FUNCTION_BLOCK TestSuite
VAR_GENERIC CONSTANT
	_MaxTestCount : DINT := 10;
END_VAR IMPLEMENTS I_TestSuite
VAR
	_TestSuiteName	  : STRING;
	TestCollection	  : ARRAY[0.._MaxTestCount] OF Test;
	NoAction		  : Test := (TestId := 'No Action', State := E_TestStatus.DoneOk);
	ActiveTest		  : DINT;
	DoneMessage		  : FB_TcMessage;
	Source			  : FB_TcSourceInfo;
	TotalTestCount	  : UDINT := 0;
	TotalOkTestCount  : UDINT := 0;
	TotalNokTestCount : UDINT := 0;
	Complete		  : BOOL;
	ResultFile		  : I_UnitTestResultFile;
	_ResultFileAdded  : BOOL;
	CurrentCycle	  : UDINT;
	Stopwatch		  : Stopwatch;
	_TestOverflowCount : UDINT;
END_VAR

{attribute 'monitoring' := 'call'}
PROPERTY Duration : LREAL
GET
Duration := Stopwatch.Elapsed;
END_GET
END_PROPERTY

//FB_Init is always available implicitly and it is used primarily for initialization.

//The return value is not evaluated. For a specific influence, you can also declare the

//methods explicitly and provide additional code there with the standard initialization

//code. You can evaluate the return value.
METHOD FB_Init : BOOL
VAR_INPUT
	bInitRetains : BOOL; // TRUE: the retain variables are initialized (reset warm / reset cold)
	bInCopyCode	 : BOOL; // TRUE: the instance will be copied to the copy code afterward (online change)
	ResultFile	 : I_UnitTestResultFile;
END_VAR
IF ResultFile <> 0 THEN
	THIS^.ResultFile := ResultFile;
END_IF
END_METHOD

{attribute 'TcRpcEnable':='1'}
METHOD ReRunIndividualTest
VAR_INPUT
	TestId : T_MaxString;
END_VAR

VAR
	i : DINT;
END_VAR
FOR i := 0 TO _MaxTestCount DO
	IF TestCollection[i].TestId = TestId THEN
		TestCollection[i].State := E_TestStatus.Init;
		ActiveTest := i;
		Complete := FALSE;
		EXIT;
	END_IF
END_FOR
END_METHOD

{attribute 'TcRpcEnable':='1'}
METHOD ReRunTests
VAR
	i : DINT;
END_VAR
FOR i := 0 TO TestSuiteParameter.MaxTestCount DO
	TestCollection[i].State := E_TestStatus.Init;
	ActiveTest				:= 0;
	Complete				:= FALSE;
	ResultFile.Initialize();
	Stopwatch.Start();
	ResultFile.AddTestSuite(Name := _TestSuiteName);
END_FOR
END_METHOD

PROPERTY ResultFileFunction : I_UnitTestResultFile
SET
ResultFile := ResultFileFunction;
END_SET
END_PROPERTY

METHOD Test : I_TestOperation
VAR_INPUT
	TestId : T_MaxString;
END_VAR

VAR
	ResultString : T_MaxString;
	i			 : DINT;
END_VAR
IF _TestSuiteName = '' THEN
	_TestSuiteName := __POUNAME();
END_IF

IF NOT _ResultFileAdded THEN
	_ResultFileAdded := TRUE;
	ResultFile.Initialize();
	Stopwatch.Start();
	ResultFile.AddTestSuite(Name := _TestSuiteName);
END_IF

IF TwinCAT_SystemInfoVarList._TaskInfo[GETCURTASKINDEXEX()].CycleCount <> CurrentCycle THEN
	CurrentCycle := TwinCAT_SystemInfoVarList._TaskInfo[GETCURTASKINDEXEX()].CycleCount;
	ResultFile.Cyclic();
END_IF

IF NOT Complete THEN
	FOR i := 0 TO _MaxTestCount DO
		TestCollection[i].TestSuiteName		 := _TestSuiteName;
		TestCollection[i].ResultFileFunction := ResultFile;
		// Detect first running test
		IF TestCollection[i].State = E_TestStatus.Running THEN
			ActiveTest := i;
		END_IF

		IF TestCollection[ActiveTest].State >= E_TestStatus.DoneOk THEN
			ActiveTest := 0;
		END_IF

		// Get existing Test
		IF (TestCollection[i].TestId = TestId) THEN
			IF (ActiveTest = i) OR (ActiveTest = 0) THEN
				Test := TestCollection[i];
			ELSE
				Test := NoAction;
			END_IF

			EXIT;
		END_IF

		// Add Test
		IF TestCollection[i].TestId = '' THEN
			TestCollection[i].TestId := TestId;
			Test					 := NoAction;
			EXIT;
		END_IF

		// Out of tests
		IF i = _MaxTestCount THEN
			Test			   := NoAction;
			_TestOverflowCount := _TestOverflowCount + 1;
			Source.sName	   := _TestSuiteName;
			DoneMessage.Create(eventClass	:= TC_EVENT_CLASSES.TestEvents,
							   nEventId		:= 1,
							   eSeverity	:= TcEventSeverity.Error,
							   ipSourceInfo := Source);

			ResultString := CONCAT('Test not added, max Tests exeeded - ', TO_STRING(_MaxTestCount));
			DoneMessage.ipArguments.AddString(ResultString);
			DoneMessage.Send(0);
			Source.Clear();
			DoneMessage.Release();
			Complete := TRUE;
		END_IF
	END_FOR

	// Run Statistic
	TotalTestCount	  := 0;
	TotalOkTestCount  := 0;
	TotalNokTestCount := 0;
	FOR i := 0 TO _MaxTestCount DO
		IF TestCollection[i].TestId <> '' THEN
			TotalTestCount := TotalTestCount + 1;
			IF TestCollection[i].State = E_TestStatus.DoneOk THEN
				TotalOkTestCount := TotalOkTestCount + 1;
			END_IF

			IF TestCollection[i].State = E_TestStatus.DoneFailed THEN
				TotalNokTestCount := TotalNokTestCount + 1;
			END_IF
		END_IF
	END_FOR

	// Tests finished
	IF (TotalTestCount = (TotalOkTestCount + TotalNokTestCount)) AND NOT Complete THEN
		Source.sName := _TestSuiteName;
		DoneMessage.Create(eventClass	:= TC_EVENT_CLASSES.TestEvents,
						   nEventId		:= 1,
						   eSeverity	:= TcEventSeverity.Error,
						   ipSourceInfo := Source);

		ResultString := CONCAT('Completed - ', CONCAT('Total Tests - ', TO_STRING(TotalTestCount)));
		ResultString := CONCAT(ResultString, CONCAT(', OK Tests - ', TO_STRING(TotalOkTestCount)));
		ResultString := CONCAT(ResultString, CONCAT(', Failed Tests - ', TO_STRING(TotalNokTestCount)));
		DoneMessage.ipArguments.AddString(ResultString);
		DoneMessage.Send(0);
		Source.Clear();
		DoneMessage.Release();

		//
		Stopwatch.Stop();
		ResultFile.AddTestSuiteStatistics(Name := _TestSuiteName, Tests := TotalTestCount, Failures := TotalNokTestCount, Duration := Stopwatch.Elapsed);
		ResultFile.SaveResult();

		//
		Complete := TRUE;
	END_IF
ELSE
	Test := NoAction;
END_IF
END_METHOD

{attribute 'monitoring' := 'call'}
PROPERTY TestOverflowCount : UDINT
GET
TestOverflowCount := _TestOverflowCount;
END_GET
END_PROPERTY

{attribute 'monitoring' := 'call'}
PROPERTY TestSuiteName : STRING
SET
_TestSuiteName := TestSuiteName;
END_SET
END_PROPERTY

END_FUNCTION_BLOCK

(* stored: Version 1.1.0.1
   POU TestSuite: Id {d93a9aa9-034f-4b1b-8d51-f63a960f5d15}, SpecialFunc None
   Property Duration: Id {7bbb8cbd-2e8a-4da3-8535-e61b5755fdb4}
   Get Get: Id {b6553703-1f1d-4dc2-bf9d-f21ab7e15224}
   Method FB_Init: Id {d564e65c-6f31-426e-ab10-2c7d7fc7cf41}
   Method ReRunIndividualTest: Id {62f6cae7-bfe8-4b44-a2ef-a751a8e71733}
   Method ReRunTests: Id {149633ad-ed2c-4a71-a7a5-f2bfddf8a7a2}
   Property ResultFileFunction: Id {2fc49ca5-ef03-4f26-b851-3c82ac31a69b}
   Set Set: Id {951f423d-d7b7-4d8b-85e2-a1939c4e8331}
   Method Test: Id {ed26b7b3-1fa1-4dc2-9f0d-d0fab78d1679}
   Property TestOverflowCount: Id {4d5e6f70-8192-4a03-8b1c-2d3e4f506172}
   Get Get: Id {5e6f7081-9203-4a14-9c2d-3e4f50617283}
   Property TestSuiteName: Id {f585ae52-04ec-4c7c-ae12-2980c5f2d3ed}
   Set Set: Id {7a5fbab5-b375-4a82-a951-31e34b901e54} *)
